{attribute 'qualified_only'}
{attribute 'strict'}
TYPE ComparisonOperator :
(
	Equal,
	NotEqual,
	LessThan,
	LessThanOrEqual,
	GreaterThan,
	GreaterThanOrEqual
);
END_TYPE

(* stored: Version 1.1.0.1
   DUT ComparisonOperator: Id {2c0f6891-5dc1-00a5-0026-68568e6fbfd7} *)
